Yaskawa INFORM job: CLEAN-R1_KM2.JBI

/JOB
//NAME CLEAN-R1_KM2
///FOLDERNAME CLEAN
//POS
///NPOS 20,20,0,0,0,0
///TOOL 0
///POSTYPE PULSE
///PULSE
C00000=2508,0,0,0,0,4169
C00001=32571,-80067,-84751,-11816,58952,90735
C00002=41115,93452,-30342,-19926,115521,85678
C00003=28599,109925,-13759,-12658,112881,84157
C00004=28301,105457,-14309,-12299,110948,84323
C00005=28966,99224,-20084,-13542,107459,84155
C00006=29027,99166,-20392,-13590,107618,84144
C00007=28599,108424,-14443,-12622,112541,84195
C00008=34011,109773,-12073,-16636,107751,84808
C00009=32816,112629,-5671,-14598,109695,85231
C00010=32618,110353,-5730,-14378,108579,85337
C00011=32545,109523,-5728,-14298,108158,85375
C00012=32618,110353,-5730,-14378,108579,85337
C00013=32816,112629,-5671,-14598,109695,85231
C00014=34011,109773,-12073,-16636,107751,84808
C00015=38810,111241,-7992,-19438,105697,85727
C00016=36913,114349,813,-16982,106196,86149
C00017=37169,116704,797,-17245,107389,86018
C00018=39968,92120,-23778,-21749,94252,85800
C00019=46315,71110,-54300,-23622,119041,85704
BC00000=0,0,0
BC00001=204899,578,1049510
BC00002=204899,578,1075157
BC00003=204899,578,1075157
BC00004=204899,578,1075157
BC00005=204899,578,1075157
BC00006=204899,578,1075157
BC00007=204899,578,1075157
BC00008=204899,578,1075157
BC00009=204899,578,1075157
BC00010=204899,578,1075157
BC00011=204899,578,1075157
BC00012=204899,578,1075157
BC00013=204899,578,1075157
BC00014=204899,578,1075157
BC00015=204899,578,1075157
BC00016=204894,578,1075156
BC00017=204894,578,1075156
BC00018=204894,578,1075156
BC00019=204899,578,1075157
//INST
///DATE 2024/04/16 12:44
///ATTR SC,RW
///GROUP1 RB1,BS1
///LVARS 0,5,0,0,0,3,3,0
NOP
SFTOF
SFTOF3D
'********************************
'Please check position before
'running in play-mode
'********************************
'#Output - Cleaning Motor
SET LI000 14
'#Output - Cleaning Oil
SET LI001 15
'#Output - Wirecut
SET LI002 16
'#Output - Wirefeeder Forward
SET LI003 4095
'#Output - Torch Blow out
SET LI004 4091
'********************************
REFP 1 C00000 BC00000
GETS LPX001 $PX011
CNVRT LPX001 LPX001 RF
GETS LPX002 $PX001
CNVRT LPX002 LPX002 RF
SUB LBP002 LBP001
'Comment out axis to shift
SETE LBP002 (1) 0
COMM SETE LBP002 (2) 0
SETE LBP002 (3) 0
SFTON LBP002
'********************************
'SAFE POS
PAUSE IF IN#(1563)=OFF
MOVJ C00001 BC00001 VJ=15.00
MOVJ C00002 BC00002 VJ=15.00
'WIRECUT
MOVJ C00003 BC00003 VJ=15.00
'WIREFEED OUTPUT
PULSE OT#(LI003) T=0.90
MOVL C00004 BC00004 V=75.0
MOVL C00005 BC00005 V=20.0
TIMER T=0.70
DOUT OT#(LI002) ON
TIMER T=1.00
MOVL C00006 BC00006 V=20.0
MOVL C00007 BC00007 V=75.0
DOUT OT#(LI002) OFF
'CLEANING MOTOR
MOVJ C00008 BC00008 VJ=50.00
MOVL C00009 BC00009 V=75.0
'CLEANING AIR
DOUT OT#(LI004) ON
MOVL C00010 BC00010 V=20.0
TIMER T=0.20
DOUT OT#(LI000) ON
TIMER T=0.50
MOVL C00011 BC00011 V=20.0
TIMER T=0.50
MOVL C00012 BC00012 V=20.0
TIMER T=0.20
DOUT OT#(LI000) OFF
TIMER T=0.50
DOUT OT#(LI004) OFF
MOVL C00013 BC00013 V=20.0
MOVL C00014 BC00014 V=75.0
'CLEANING OIL
MOVJ C00015 BC00015 VJ=50.00
MOVL C00016 BC00016 V=75.0
PULSE OT#(LI001) T=0.20
TIMER T=1.00
MOVL C00017 BC00017 V=75.0
'CLEANING AIR
PULSE OT#(LI004) T=1.00
TIMER T=1.00
MOVJ C00018 BC00018 VJ=25.00
'SAFE POS
MOVJ C00019 BC00019 VJ=15.00
SFTOF
'********************************
'*         CLEANING JOB         *
'*      __ __ _____ _____       *
'*     |  |  |   | | __  |      *
'*     |_   _| | | |    -|      *
'*       |_| |_|___|__|__|      *
'*        YRC Multi Base        *
'*       rev 4. 2021-10-12      *
'********************************
END
